INTERFACE I_MessageData

PROPERTY DirRoot : POINTER to string(255)
SET
END_SET
END_PROPERTY

PROPERTY ErrorIndex : reference to uint
SET
END_SET
END_PROPERTY

PROPERTY FileRoot : pointer to string(255)
SET
END_SET
END_PROPERTY

PROPERTY LocalTime : pointer to DT
SET
END_SET
END_PROPERTY

PROPERTY MessageIndex : reference to uint
SET
END_SET
END_PROPERTY

PROPERTY MsgList : pointer to ARRAY[1..GVL_MSG.MAX_MESSAGE] OF st_message
SET
END_SET
END_PROPERTY

END_INTERFACE

(* stored: Version 1.1.0.1, ProductVersion 3.1.4026.18
   Itf I_MessageData: Id {d6f693ca-67bb-4cc0-ba34-ba7db9d27673}
   Property DirRoot: Id {4200c488-1d8a-46ce-8d59-26a9cc9e84e0}
   Set Set: Id {bd8eca24-23c0-427b-8763-5ac2e21d12de}
   Property ErrorIndex: Id {546a555b-3af5-4614-9d72-29d965252edd}
   Set Set: Id {6e883f9e-3a5f-432b-a123-ff13252eccc4}
   Property FileRoot: Id {45a2813e-a4a2-4d96-b7a2-58468f177462}
   Set Set: Id {4c3e5f81-27e0-4806-9f85-f997c1826008}
   Property LocalTime: Id {bbcf7938-fe42-49f8-8b28-cd822d01c334}
   Set Set: Id {d45fe9a1-2715-432e-957a-be1fe5d27556}
   Property MessageIndex: Id {ac687701-88e8-4108-a7d1-9d1cb5705c76}
   Set Set: Id {a5863ddd-91b0-4254-a5ce-dfe43580fc63}
   Property MsgList: Id {41396092-862a-4bca-88a9-16ef870f3b18}
   Set Set: Id {b0202562-d01d-45c9-9d08-1ab1ec2c9272} *)
